// TIA Portal V17 export
FUNCTION "FC_FanGasControl" : Void   // FC, LAD
{ S7_Optimized_Access := 'TRUE' }
BEGIN

REGION Network 1: 风机运行联锁
   // 风机运行按接通且风机故障反馈未动作时，驱动风机运行线圈
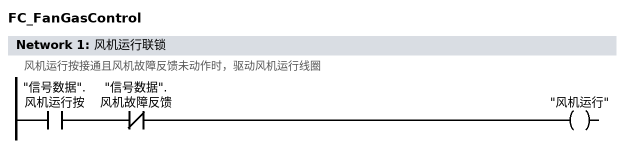
   RUNG wire#powerrail
      Contact( "信号数据".风机运行按 )
      I_Contact( "信号数据".风机故障反馈 )
      Coil( "风机运行" )
   END_RUNG
   // the same network as SCL:
   "风机运行" := "信号数据".风机运行按 AND NOT "信号数据".风机故障反馈;
END_REGION
END_FUNCTION
